// TIA Portal V17 export
// export: Created 2022-04-06T07:28:40.9307811Z, ExportSetting WithDefaults, DisplayName Totally Integrated Automation Portal, DisplayVersion V17, DisplayName TIA Portal Openness, DisplayVersion V17, DisplayName TIA Portal Version Control Interface, DisplayVersion V17, DisplayName TIA Portal Test Suite Advanced, DisplayVersion V17, DisplayName SINAMICS Startdrive Advanced, DisplayVersion V17, DisplayName SINAMICS Startdrive G130, G150, S120, S150, SINAMICS MV, S210, DisplayVersion V17, DisplayName SINAMICS Startdrive G110M, G120, G120C, G120D, G120P, G115D, DisplayVersion V17, DisplayName STEP 7 Professional, DisplayVersion V17, DisplayName STEP 7 Safety, DisplayVersion V17, DisplayName WinCC Advanced / Unified PC, DisplayVersion V17
TYPE "LAxisCtrl_typeDiagnostics"
TITLE = LAxisCtrl_typeDiagnostics
// Support: tech.team.motioncontrol@siemens.com
// stored: IsFailsafeCompliant false
   STRUCT
      status { ExternalWritable := 'False'} : Word := 16#0000;   // Status of FB when error occurred
      subfunctionStatus { ExternalWritable := 'False'} : Word := 16#0000;   // ErrorID of called subfunction
      basicMotionState { ExternalWritable := 'False'} : DInt := 0;   // Current basic motion state when error occurred
      superimposedMotionState { ExternalWritable := 'False'} : DInt := 0;   // Current superimposed motion state when error occurred
   END_STRUCT;
END_TYPE
